TYPE st_PLCtoHMI_Robot :
STRUCT
    state : eState;
END_STRUCT
END_TYPE

(* stored: Version 1.1.0.1, ProductVersion 3.1.4024.9
   DUT st_PLCtoHMI_Robot: Id {bc0c60ad-ba30-41e5-a6e8-b04dc8e2f4b9} *)
